{attribute 'qualified_only'}
{attribute 'strict'}
{attribute 'to_string'}
TYPE cLaneSel :
(
	None := 0,
	Green := 1,
	Red := 2,
	Blue := 3
);
END_TYPE

(* stored: Version 1.1.0.1, ProductVersion 3.1.4024.6
   DUT cLaneSel: Id {7a8c9d0c-2b25-4fa7-a0b0-f40d91157b7e} *)
